// TIA Portal project "Tisch" (V17)

(* hardware
DEVICE "S7-1200-Station_2"  S7-1200 Station
   slot 0: "Baugruppenträger_0"  S7-1200 Rack  Rack  V1.0
   slot 1: "MTLab2-SPS-11"  CPU 1215C AC/DC/Rly  6ES7 215-1BG40-0XB0  V4.5
   slot 2: "DI 16/DQ 16x24VDC_1"  SM 1223 DI16/DQ16 x 24VDC  6ES7 223-1BL30-0XB0  V1.0
   slot 3: "DI 16/DQ 16x24VDC_2"  SM 1223 DI16/DQ16 x 24VDC  6ES7 223-1BL30-0XB0  V1.0
   slot 4: "AI 4x13BIT/AQ 2x14BIT_1"  SM 1234 AI4/AQ2  6ES7 234-4HE30-0XB0  V1.0
*)

// ===== PLC "MTLab2-SPS-11"  CPU 1215C AC/DC/Rly =====

VAR_GLOBAL   // PLC tag table "io_Tisch2_alt_Dreharm"
   "di_Encoder_ChA" AT %I0.0 : Bool;
   "di_Encoder_ChB" AT %I0.1 : Bool;
   "di_0Deg_Position" AT %I0.2 : Bool;
   "d_Z-Achse_ist_eingefahren" AT %I0.3 : Bool;
   "di_Z-Achse_ist_ausgefahren" AT %I0.4 : Bool;
   "di_Vertikalzylinder_ist_unten" AT %I0.5 : Bool;
   "di_Vertikalzylinder_ist_oben" AT %I0.6 : Bool;
   "do_Vertikalzylinder_nach_oben" AT %Q0.0 : Bool;
   "do_Sauger_ein" AT %Q0.1 : Bool;
   "do_Z-Achse_ausfahren" AT %Q0.2 : Bool;
   "do_drehen_links" AT %Q0.3 : Bool;
   "do_drehen_rechts" AT %Q0.4 : Bool;
   "di_Drehgeber_Wert" AT %ID1000 : DInt;
END_VAR

VAR_GLOBAL   // PLC tag table "io_Tisch2_alt_Förderband"
   "di_Lichtschranke" AT %E13.4 : Bool;
   "do_Rechtslauf" AT %A13.0 : Bool;
   "do_Linkslauf" AT %A13.1 : Bool;
END_VAR

VAR_GLOBAL   // PLC tag table "io_Tisch2_alt_Portal"
   "di_Zylinder_ist_oben" AT %E13.0 : Bool;
   "di_Zylinder_ist_unten" AT %E13.1 : Bool;
   "di_Shuttle_ist_rechts" AT %I13.2 : Bool;
   "di_Shuttle_ist_links" AT %I13.3 : Bool;
   "do_Zylinder_runter" AT %A8.4 : Bool;
   "do_Shuttle_links" AT %Q8.5 : Bool;
   "do_Saugen_ein" AT %Q8.6 : Bool;
END_VAR

VAR_GLOBAL   // PLC tag table "io_Tisch2_alt_Presse"
   "di_Sicherheitstür_ist_oben(1)" AT %E12.0 : Bool;
   "di_Sicherheitstür_ist_unten(1)" AT %E12.1 : Bool;
   "di_Ausschub_ist_ausgefahren(1)" AT %E12.2 : Bool;
   "di_Ausschub_ist_eingefahren(1)" AT %E12.3 : Bool;
   "di_Taster_rechts" AT %E12.4 : Bool;
   "di_Taster_links" AT %E12.5 : Bool;
   "do_Sicherheitstür_öffnen(1)" AT %A12.0 : Bool;
   "do_Sicherheitstür_schliessen(1)" AT %A12.1 : Bool;
   "do_Ausschub_ausfahren(1)" AT %A12.2 : Bool;
   "do_Ausschub_einfahren(1)" AT %A12.3 : Bool;
   "do_Lampe_rechts" AT %A12.4 : Bool;
   "do_Lampe_links" AT %A12.5 : Bool;
   "do_Stempel_senken(1)" AT %A12.6 : Bool;
   "do_Stempel_heben(1)" AT %A12.7 : Bool;
END_VAR

VAR_GLOBAL   // PLC tag table "io_Tisch2_alt_Stiftstation"
   "di_Klemmzylinder_ist_ausgefahren" AT %E1.1 : Bool;
   "di_Klemmzylinder_ist_eingefahren" AT %E1.2 : Bool;
   "di_Stiftzylinder_ist_ausgefahren" AT %E1.3 : Bool;
   "di_Stiftzylinder_ist_eingefahren" AT %E1.4 : Bool;
   "do_Klemmzylinder_ausfahren" AT %A0.7 : Bool;
   "do_Stiftzylinder_ausfahren" AT %A1.0 : Bool;
END_VAR

VAR_GLOBAL   // PLC tag table "io_Tisch2_alt_Bedienpult"
   "di_NotAus(NC)(1)" AT %E8.0 : Bool;
   "di_Hand(1)" AT %E8.1 : Bool;
   "di_Auto(1)" AT %E8.2 : Bool;
   "di_Start(1)" AT %E8.3 : Bool;
   "di_Stop(1)" AT %E8.4 : Bool;
   "di_Quit(1)" AT %E8.5 : Bool;
   "di_S6" AT %E8.6 : Bool;
   "di_NotAus(NO)" AT %E8.7 : Bool;
   "di_S1(1)" AT %E9.0 : Bool;
   "di_S2(1)" AT %E9.1 : Bool;
   "di_S3" AT %E9.2 : Bool;
   "di_S4" AT %E9.3 : Bool;
   "di_S5" AT %E9.4 : Bool;
   "do_Meldeleuchte_Bereit" AT %A8.0 : Bool;
   "do_Meldeleuchte_Läuft" AT %A8.1 : Bool;
   "do_Meldeleuchte_Fehler" AT %A8.2 : Bool;
   "do_Meldeleuchte_S6" AT %A8.3 : Bool;
END_VAR

TYPE "Type_Anlage"
   STRUCT
      Modus : Struct
         Grundstellung : Bool;
         Auto : Bool;
         Hand : Bool;
      END_STRUCT;
      NotHalt : Bool;
   END_STRUCT;
END_TYPE

TYPE "Type_Modul"
   STRUCT
      Kommando : Struct
         Start : Bool;
      END_STRUCT;
      Status : Struct
         Bereit : Bool;
         Fehler : Bool;
         LED : Bool;
      END_STRUCT;
      Parameter : Struct
         LongPressHomePosition : Time := T#2s;
      END_STRUCT;
   END_STRUCT;
END_TYPE

// folder: 1_DB

DATA_BLOCK "DB_Anlage"   // DB4
{ S7_Optimized_Access := 'TRUE' }
VERSION : 0.1
BEGIN
END_DATA_BLOCK

// folder: 8_Hardware/Aktoren

DATA_BLOCK "PortalLinks"   // DB25
{ S7_Optimized_Access := 'TRUE' }
VERSION : 0.1
// stored: InstanceOfName FB_SCL_Aktor
"FB_SCL_Aktor"
BEGIN
END_DATA_BLOCK

// folder: 8_Hardware/Sensoren

DATA_BLOCK "Starttaster"   // DB1
{ S7_Optimized_Access := 'TRUE' }
VERSION : 0.1
// stored: InstanceOfName FB_SCL_Sensor
"FB_SCL_Sensor"
BEGIN
END_DATA_BLOCK

DATA_BLOCK "Handmodus"   // DB2
{ S7_Optimized_Access := 'TRUE' }
VERSION : 0.1
// stored: InstanceOfName FB_SCL_Sensor
"FB_SCL_Sensor"
BEGIN
END_DATA_BLOCK

DATA_BLOCK "Automodus"   // DB3
{ S7_Optimized_Access := 'TRUE' }
VERSION : 0.1
// stored: InstanceOfName FB_SCL_Sensor
"FB_SCL_Sensor"
BEGIN
END_DATA_BLOCK

DATA_BLOCK "Grundstellung"   // DB5
{ S7_Optimized_Access := 'TRUE' }
VERSION : 0.1
// stored: InstanceOfName FB_SCL_Sensor
"FB_SCL_Sensor"
BEGIN
END_DATA_BLOCK

DATA_BLOCK "PortalBandseitig"   // DB21
{ S7_Optimized_Access := 'TRUE' }
VERSION : 0.1
// stored: InstanceOfName FB_SCL_Sensor
"FB_SCL_Sensor"
BEGIN
END_DATA_BLOCK

DATA_BLOCK "PortalPressenseitig"   // DB22
{ S7_Optimized_Access := 'TRUE' }
VERSION : 0.1
// stored: InstanceOfName FB_SCL_Sensor
"FB_SCL_Sensor"
BEGIN
END_DATA_BLOCK

DATA_BLOCK "PortalOben"   // DB23
{ S7_Optimized_Access := 'TRUE' }
VERSION : 0.1
// stored: InstanceOfName FB_SCL_Sensor
"FB_SCL_Sensor"
BEGIN
END_DATA_BLOCK

DATA_BLOCK "PortalUnten"   // DB24
{ S7_Optimized_Access := 'TRUE' }
VERSION : 0.1
// stored: InstanceOfName FB_SCL_Sensor
"FB_SCL_Sensor"
BEGIN
END_DATA_BLOCK

// folder: 8_Hardware/Zylinder

DATA_BLOCK "TestZylinder_1V2ES"   // DB20
{ S7_Optimized_Access := 'TRUE' }
VERSION : 0.1
// stored: InstanceOfName 1_FB_SCL_Zylinder_1V_2ES
"1_FB_SCL_Zylinder_1V_2ES"
BEGIN
END_DATA_BLOCK

// folder: 1_DB

FUNCTION "FC_Bedienpult" : Void   // FC4, FBD
{ S7_Optimized_Access := 'TRUE' }
VERSION : 0.1
BEGIN

REGION Network 1
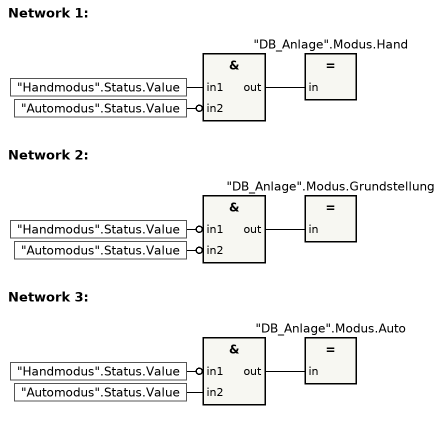
   "DB_Anlage".Modus.Hand := "Handmodus".Status.Value AND NOT "Automodus".Status.Value;
END_REGION

REGION Network 2
   "DB_Anlage".Modus.Grundstellung := NOT "Handmodus".Status.Value AND NOT "Automodus".Status.Value;
END_REGION

REGION Network 3
   "DB_Anlage".Modus.Auto := NOT "Handmodus".Status.Value AND "Automodus".Status.Value;
END_REGION
END_FUNCTION

ORGANIZATION_BLOCK "Main_DB"   // OB124, FBD, ProgramCycle
TITLE = "Main Program Sweep (Cycle)"
{ S7_Optimized_Access := 'TRUE' }
VERSION : 0.1
BEGIN

REGION Network 1: Variablen von/zum HMI aktualisieren
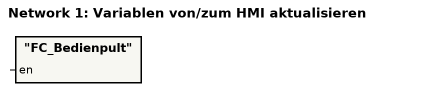
   "FC_Bedienpult"();
END_REGION
END_ORGANIZATION_BLOCK

// folder: 2_Ablauf/1_Module/4_Presse

FUNCTION_BLOCK "FB_SCL_Ablauf_Presse"   // FB8, SCL
{ S7_Optimized_Access := 'TRUE' }
VERSION : 0.1
   VAR_IN_OUT
      Zylinder_Ausschub : "0_FB_SCL_Zylinder_2V_2ES";
      Zylinder_Sicherheitstüre : "0_FB_SCL_Zylinder_2V_2ES";
      Zylinder_Presse : "0_FB_SCL_Zylinder_2V_2ES";
   END_VAR
   VAR
      homePosition : Bool;
      previousState : Int;
      currentState : Int;
      nextState : Int;
      stateStartTimeMs : UDInt;
      Kommando : Struct
         AutomatikStart : Bool;
         HomePositionStart : Bool;
         Retry : Bool;
      END_STRUCT;
      Status : Struct
         Ready : Bool;
         Error : Bool;
      END_STRUCT;
   END_VAR
   VAR_TEMP
      currentTimeMs : UDInt;
      stateActiveTimeS : UDInt;
      stateActiveTimeMs : UDInt;
   END_VAR
   VAR CONSTANT
      STATE_INIT : Int;
      STATE_READY : Int := 1;
      STATE_AUTO_FINISHED : Int := 2;
      STATE_AUTO_MOVE1 : Int := 3;
      STATE_HOMEPOSITION_FINISHED : Int := 4;
      STATE_HOMEPOSITION_MOVE1 : Int := 5;
      STATE_ERROR : Int := 6;
   END_VAR
BEGIN
   REGION State Machine Control
       // get current time
       "getTimestamp"(#currentTimeMs);

       REGION State Transition Check
           // check if a state transition is neccessary and store the time
           IF (#nextState <> #currentState) THEN
               // state transition occured!
               #previousState := #currentState;
               #currentState := #nextState;        // activate the new state
               #stateStartTimeMs := #currentTimeMs;  // store the time when the state was activated
           END_IF;
       END_REGION

       // calculate the time the state is already active
       #stateActiveTimeMs := #currentTimeMs - #stateStartTimeMs;
       #stateActiveTimeS := #stateActiveTimeMs / 1000;
   END_REGION


   // a move to startPosition request is executed regardless of the current state
   IF (#Kommando.HomePositionStart) THEN
       #nextState := #STATE_HOMEPOSITION_MOVE1;
   END_IF;

   REGION CASE Structure

       CASE #currentState OF


               // first state after machine startup
           #STATE_INIT:
               // set outputs to default values
               #Status.Ready := false;
               #Status.Error := false;

               // check if system is in "Grundstellung"
               IF (#homePosition) THEN
                   #nextState := #STATE_READY;
               END_IF;



           #STATE_READY:
               // system is ready to start
               #Status.Ready := true;

               // wait until rising edge of start signal occurs
               IF (#Kommando.AutomatikStart) THEN
                   #Status.Ready := false;
                   #nextState := #STATE_AUTO_MOVE1;
               END_IF;

           #STATE_AUTO_FINISHED:
               #nextState := #STATE_INIT;

           #STATE_HOMEPOSITION_FINISHED:
               #nextState := #STATE_INIT;




           #STATE_AUTO_MOVE1:
               // do something
               // 

               // if finished then goto finished
               #nextState := #STATE_AUTO_FINISHED;

               // transition to other states only if #DB_Anlage.Status.Auto_Aktiv is true!

           #STATE_HOMEPOSITION_MOVE1:
               // do something

               // if finished then goto finished
               #nextState := #STATE_HOMEPOSITION_FINISHED;

               // transition to other states only if #DB_Anlage.Status.Grundstellung_Aktiv is true!



           #STATE_ERROR:
               #Status.Ready := false;
               #Status.Error := true;

               // wait until the user has removed the error source
               IF (#Kommando.Retry) THEN
                   // go back to the last state and retry
                   #nextState := #previousState;
               END_IF;

       END_CASE;
   END_REGION

   // input signals are only true for one cycle
   #Kommando.AutomatikStart := false;
   #Kommando.HomePositionStart := false;
   #Kommando.Retry := false;
END_FUNCTION_BLOCK

// folder: 8_Hardware

FUNCTION "FC_Zylinder" : Void   // FC1, FBD
{ S7_Optimized_Access := 'TRUE' }
VERSION : 0.1
// hier werden den Zylindern die Ein- und Ausgänge zugewiesen
BEGIN

REGION Network 1
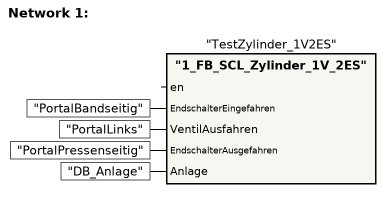
   "TestZylinder_1V2ES"(EndschalterEingefahren := "PortalBandseitig",   // "1_FB_SCL_Zylinder_1V_2ES"
                        VentilAusfahren := "PortalLinks",
                        EndschalterAusgefahren := "PortalPressenseitig",
                        Anlage := "DB_Anlage");
END_REGION
END_FUNCTION

FUNCTION "FC_Aktoren" : Void   // FC2, FBD
{ S7_Optimized_Access := 'TRUE' }
VERSION : 0.1
BEGIN

REGION Network 1
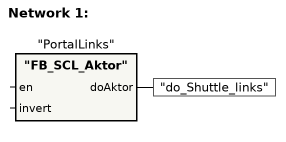
   "PortalLinks"(doAktor => "do_Shuttle_links");   // "FB_SCL_Aktor"
END_REGION
END_FUNCTION

FUNCTION "FC_Sensor" : Void   // FC3, FBD
{ S7_Optimized_Access := 'TRUE' }
VERSION : 0.1
BEGIN

REGION Network 1
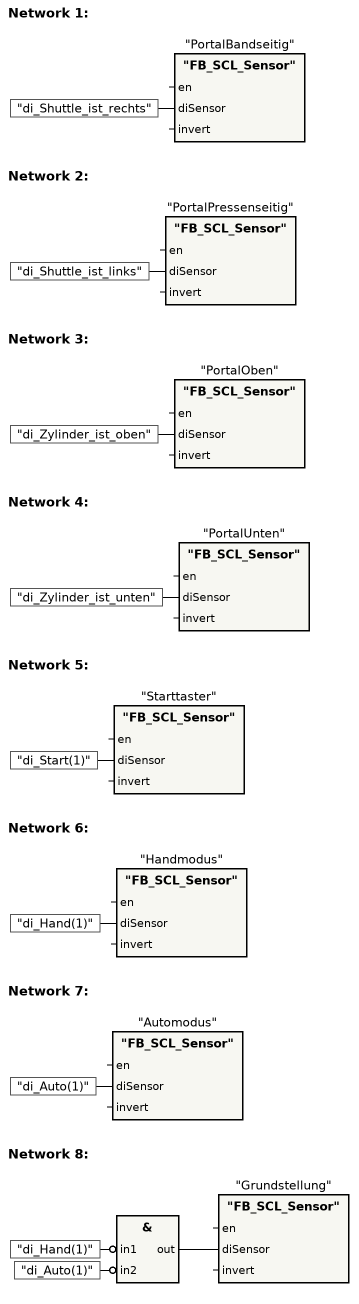
   "PortalBandseitig"(diSensor := "di_Shuttle_ist_rechts");   // "FB_SCL_Sensor"
END_REGION

REGION Network 2
   "PortalPressenseitig"(diSensor := "di_Shuttle_ist_links");   // "FB_SCL_Sensor"
END_REGION

REGION Network 3
   "PortalOben"(diSensor := "di_Zylinder_ist_oben");   // "FB_SCL_Sensor"
END_REGION

REGION Network 4
   "PortalUnten"(diSensor := "di_Zylinder_ist_unten");   // "FB_SCL_Sensor"
END_REGION

REGION Network 5
   "Starttaster"(diSensor := "di_Start(1)");   // "FB_SCL_Sensor"
END_REGION

REGION Network 6
   "Handmodus"(diSensor := "di_Hand(1)");   // "FB_SCL_Sensor"
END_REGION

REGION Network 7
   "Automodus"(diSensor := "di_Auto(1)");   // "FB_SCL_Sensor"
END_REGION

REGION Network 8
   "Grundstellung"(diSensor := NOT "di_Hand(1)" AND NOT "di_Auto(1)");   // "FB_SCL_Sensor"
END_REGION
END_FUNCTION

ORGANIZATION_BLOCK "Main_Hardware"   // OB123, FBD, ProgramCycle
TITLE = "Main Program Sweep (Cycle)"
{ S7_Optimized_Access := 'TRUE' }
VERSION : 0.1
BEGIN

REGION Network 1: Motoren ansteuern
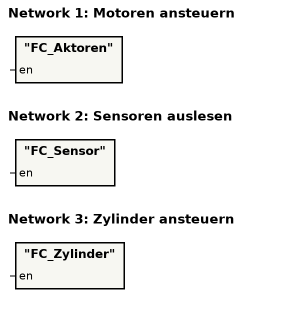
   "FC_Aktoren"();
END_REGION

REGION Network 2: Sensoren auslesen
   "FC_Sensor"();
END_REGION

REGION Network 3: Zylinder ansteuern
   "FC_Zylinder"();
END_REGION
END_ORGANIZATION_BLOCK

// folder: 9_Lib/0_Hardware/Sensor

FUNCTION_BLOCK "FB_SCL_Sensor"   // FB3, SCL
{ S7_Optimized_Access := 'TRUE' }
VERSION : 0.1
   VAR_INPUT
      diSensor : Bool;
      invert : Bool;
   END_VAR
   VAR
      Status : Struct
         Value : Bool;
      END_STRUCT;
   END_VAR
BEGIN
   IF #invert = TRUE THEN          //If Value is inverted, then return the inverted value
       #Status.Value := NOT #diSensor;
   ELSE                            //If Value is not inverted, then return the value itself
       #Status.Value := #diSensor;
   END_IF;
END_FUNCTION_BLOCK

FUNCTION_BLOCK "FB_SCL_Aktor"   // FB5, SCL
{ S7_Optimized_Access := 'TRUE' }
VERSION : 0.1
   VAR_INPUT
      invert : Bool;
   END_VAR
   VAR_OUTPUT
      doAktor : Bool;
   END_VAR
   VAR
      Kommando : Struct
         Value : Bool;
      END_STRUCT;
   END_VAR
BEGIN
   IF #invert THEN
       #doAktor := NOT #Kommando.Value;
   ELSE
       #doAktor := #Kommando.Value;
   END_IF;
END_FUNCTION_BLOCK

// folder: 9_Lib/0_Hardware/Zylinder/Varianten

FUNCTION_BLOCK "0_FB_SCL_Zylinder_2V_2ES"   // FB1, SCL
{ S7_Optimized_Access := 'TRUE' }
VERSION : 0.1
   VAR_IN_OUT
      EndschalterEingefahren : "FB_SCL_Sensor";
      VentilAusfahren : "FB_SCL_Aktor";
      VentilEinfahren : "FB_SCL_Aktor";
      EndschalterAusgefahren : "FB_SCL_Sensor";
      Anlage : "Type_Anlage";
   END_VAR
   VAR
      Status : Struct
         istAusgefahren : Bool;
         istEingefahren : Bool;
         Fehler : Bool;
         Bereit : Bool;
      END_STRUCT;
      Parameter : Struct
         timeoutEinfahrenMS : Int := 1000;
         timeoutAusfahrenMS : Int := 1000;
         ZeitDruckaufbauMS : Int := 250;
         WartezeitInitMS : Int := 250;
      END_STRUCT;
      Kommando : Struct
         einfahren : Bool;
         ausfahren : Bool;
         einzelschrittStart : Bool;
      END_STRUCT;
      StateMachine : Struct
         CurrentState : Int := 999;
         NextState : Int;
         StateStartTimeMS : UDInt;
      END_STRUCT;
   END_VAR
   VAR_TEMP
      CurrentTimeMS : UDInt;
      stateActiveTimeMS : UDInt;
   END_VAR
   VAR CONSTANT
      STATE_INIT : Int := 0;
      STATE_BUILDPRESSURE : Int := 1;
      STATE_READY : Int := 2;
      STATE_SINGLEEXTEND : Int := 3;
      STATE_EXTEND : Int := 4;
      STATE_ENDPOS : Int := 5;
      STATE_ERROR : Int := 6;
      STATE_SINGLERETRACT : Int := 7;
      STATE_RETRACT : Int := 8;
   END_VAR
BEGIN
   REGION NotHalt

       IF #Anlage.NotHalt THEN
           #VentilAusfahren.Kommando.Value := FALSE;
           #VentilEinfahren.Kommando.Value := FALSE;
           RETURN;
       END_IF;

   END_REGION

   REGION Timing
       // get current time
       "getTimestamp"(#CurrentTimeMS);


       // check if a state transition is neccessary and store the time
       IF (#StateMachine.NextState <> #StateMachine.CurrentState) THEN
           // state transition occured!
           #StateMachine.CurrentState := #StateMachine.NextState;        // activate the new state
           #StateMachine.StateStartTimeMS := #CurrentTimeMS;  // store the time when the state was activated
       END_IF;

       // calculate the time the state is already active
       #stateActiveTimeMS := #CurrentTimeMS - #StateMachine.StateStartTimeMS;
   END_REGION

   REGION Logik

       CASE #StateMachine.CurrentState OF

           #STATE_INIT:  //INIT
               REGION INIT

               IF #stateActiveTimeMS > #Parameter.WartezeitInitMS THEN
                   #StateMachine.NextState := #STATE_BUILDPRESSURE;
               END_IF;
           END_REGION

           #STATE_BUILDPRESSURE:
               REGION BUILD PRESSURE
               #Status.Fehler := FALSE;

               IF (#EndschalterAusgefahren.Status.Value AND #EndschalterEingefahren.Status.Value) OR (NOT #EndschalterAusgefahren.Status.Value AND NOT #EndschalterEingefahren.Status.Value) THEN
                   #Status.Fehler := TRUE;
                   #VentilEinfahren.Kommando.Value := false;
                   #VentilAusfahren.Kommando.Value := false;
                   #StateMachine.NextState := #STATE_READY;
               END_IF;

               IF #EndschalterAusgefahren.Status.Value AND NOT #EndschalterEingefahren.Status.Value THEN
                   #VentilAusfahren.Kommando.Value := true;
                   #VentilEinfahren.Kommando.Value := false;
               ELSIF #EndschalterEingefahren.Status.Value AND NOT #EndschalterAusgefahren.Status.Value THEN
                   #VentilAusfahren.Kommando.Value := FALSE;
                   #VentilEinfahren.Kommando.Value := TRUE;
               END_IF;

               IF #stateActiveTimeMS > #Parameter.ZeitDruckaufbauMS THEN
                   #VentilEinfahren.Kommando.Value := false;
                   #VentilAusfahren.Kommando.Value := false;
                   #StateMachine.NextState := #STATE_READY;
               END_IF;

           END_REGION

           #STATE_READY:
               REGION Ready
                   #Status.Bereit := true;
                   IF #Kommando.ausfahren AND NOT #VentilAusfahren.Kommando.Value THEN
                       #StateMachine.NextState := #STATE_SINGLEEXTEND;
                   END_IF;

                   IF #Kommando.einfahren AND NOT #EndschalterEingefahren.Status.Value THEN
                       #StateMachine.NextState := #STATE_SINGLERETRACT;
                   END_IF;

               END_REGION

           #STATE_SINGLEEXTEND:
               REGION Single Step Extension

                   #Status.Bereit := false;

                   IF NOT #Anlage.Modus.Hand THEN
                       #StateMachine.NextState := #STATE_READY;
                   END_IF;

                   IF #Anlage.Modus.Hand AND #Kommando.einzelschrittStart THEN
                       #StateMachine.NextState := #STATE_EXTEND;
                   END_IF;

                   IF #Anlage.Modus.Auto OR #Anlage.Modus.Grundstellung THEN
                       #StateMachine.NextState := #STATE_EXTEND;
                   END_IF;

               END_REGION

           #STATE_EXTEND:
               REGION Extension
                   #VentilAusfahren.Kommando.Value := true;
                   IF #EndschalterAusgefahren.Status.Value THEN
                       #StateMachine.NextState := #STATE_ENDPOS;
                   END_IF;

                   IF #stateActiveTimeMS > #Parameter.timeoutAusfahrenMS THEN
                       #StateMachine.NextState := #STATE_ERROR;
                   END_IF;
               END_REGION;

           #STATE_SINGLERETRACT:
               REGION Single Step Retract

                   #Status.Bereit := false;

                   IF NOT #Anlage.Modus.Hand THEN
                       #StateMachine.NextState := #STATE_READY;
                   END_IF;

                   IF #Anlage.Modus.Hand AND #Kommando.einzelschrittStart THEN
                       #StateMachine.NextState := #STATE_RETRACT;
                   END_IF;

                   IF #Anlage.Modus.Auto OR #Anlage.Modus.Grundstellung THEN
                       #StateMachine.NextState := #STATE_RETRACT;
                   END_IF;

               END_REGION

           #STATE_RETRACT:
               REGION Extension
                   #VentilEinfahren.Kommando.Value := true;
                   IF #EndschalterEingefahren.Status.Value THEN
                       #StateMachine.NextState := #STATE_ENDPOS;
                   END_IF;

                   IF #stateActiveTimeMS > #Parameter.timeoutEinfahrenMS THEN
                       #StateMachine.NextState := #STATE_ERROR;
                   END_IF;
               END_REGION

           #STATE_ENDPOS:
               REGION End Position
                   #VentilAusfahren.Kommando.Value := false;
                   #VentilEinfahren.Kommando.Value := false;
                   #Status.Fehler := false;
                   #StateMachine.NextState := #STATE_READY;
               END_REGION;

           #STATE_ERROR:
               REGION End Position
                   #VentilAusfahren.Kommando.Value := false;
                   #VentilEinfahren.Kommando.Value := false;
                   #Status.Fehler := true;
                   #StateMachine.NextState := #STATE_READY;
               END_REGION ;


       END_CASE;


   END_REGION

   REGION KommandoReset

       #Kommando.ausfahren := FALSE;
       #Kommando.einfahren := FALSE;
       #Kommando.einzelschrittStart := FALSE;

   END_REGION
END_FUNCTION_BLOCK

FUNCTION_BLOCK "1_FB_SCL_Zylinder_1V_2ES"   // FB2, SCL
{ S7_Optimized_Access := 'TRUE' }
VERSION : 0.1
   VAR_IN_OUT
      EndschalterEingefahren : "FB_SCL_Sensor";
      VentilAusfahren : "FB_SCL_Aktor";
      EndschalterAusgefahren : "FB_SCL_Sensor";
      Anlage : "Type_Anlage";
   END_VAR
   VAR
      Status : Struct
         istAusgefahren : Bool;
         istEingefahren : Bool;
         Fehler : Bool;
         Bereit : Bool;
      END_STRUCT;
      Parameter : Struct
         timeoutEinfahrenMS : Int := 1000;
         timeoutAusfahrenMS : Int := 1000;
         ZeitDruckaufbauMS : Int := 250;
         WartezeitInitMS : Int := 250;
      END_STRUCT;
      Kommando : Struct
         einfahren : Bool;
         ausfahren : Bool;
         einzelschrittStart : Bool;
      END_STRUCT;
      StaticOutput : Bool;   // Static Variable to set for output
      StateMachine : Struct
         CurrentState : Int := 999;
         NextState : Int;
         StateStartTimeMS : UDInt;
      END_STRUCT;
   END_VAR
   VAR_TEMP
      CurrentTimeMS : UDInt;
      stateActiveTimeMS : UDInt;
   END_VAR
   VAR CONSTANT
      STATE_INIT : Int := 0;
      STATE_BUILDPRESSURE : Int := 1;
      STATE_READY : Int := 2;
      STATE_SINGLEEXTEND : Int := 3;
      STATE_EXTEND : Int := 4;
      STATE_ENDPOS : Int := 5;
      STATE_ERROR : Int := 6;
      STATE_SINGLERETRACT : Int := 7;
      STATE_RETRACT : Int := 8;
   END_VAR
BEGIN
   //Copied code from 0_FB_SCL_Zylinder_2V_2ES,
   //Output is now a static variable ("StaticOutput"), which is written to the output at the end
   //There is no Valve for Contraction

   REGION NotHalt

       IF #Anlage.NotHalt THEN
           #VentilAusfahren.Kommando.Value := FALSE;
           RETURN;
       END_IF;

   END_REGION

   REGION Timing
       // get current time
       "getTimestamp"(#CurrentTimeMS);


       // check if a state transition is neccessary and store the time
       IF (#StateMachine.NextState <> #StateMachine.CurrentState) THEN
           // state transition occured!
           #StateMachine.CurrentState := #StateMachine.NextState;        // activate the new state
           #StateMachine.StateStartTimeMS := #CurrentTimeMS;  // store the time when the state was activated
       END_IF;

       // calculate the time the state is already active
       #stateActiveTimeMS := #CurrentTimeMS - #StateMachine.StateStartTimeMS;
   END_REGION

   REGION Logik

       CASE #StateMachine.CurrentState OF

           #STATE_INIT:  //INIT
               REGION INIT

               IF #stateActiveTimeMS > #Parameter.WartezeitInitMS THEN
                   #StateMachine.NextState := #STATE_BUILDPRESSURE;
               END_IF;
           END_REGION

           #STATE_BUILDPRESSURE:
               REGION BUILD PRESSURE
               #Status.Fehler := FALSE;

               IF (#EndschalterAusgefahren.Status.Value AND #EndschalterEingefahren.Status.Value) OR (NOT #EndschalterAusgefahren.Status.Value AND NOT #EndschalterEingefahren.Status.Value) THEN
                   #Status.Fehler := TRUE;
                   #StaticOutput := FALSE;
                   #StateMachine.NextState := #STATE_READY;
               END_IF;

               IF #EndschalterAusgefahren.Status.Value AND NOT #EndschalterEingefahren.Status.Value THEN
                   #StaticOutput := TRUE;
               ELSIF #EndschalterEingefahren.Status.Value AND NOT #EndschalterAusgefahren.Status.Value THEN
                   #StaticOutput := FALSE;
               END_IF;

               IF #stateActiveTimeMS > #Parameter.ZeitDruckaufbauMS THEN
                   #StaticOutput := FALSE;
                   #StateMachine.NextState := #STATE_READY;
               END_IF;

           END_REGION

           #STATE_READY:
               REGION Ready
                   #Status.Bereit := true;
                   IF #Kommando.ausfahren AND NOT #VentilAusfahren.Kommando.Value THEN
                       #StateMachine.NextState := #STATE_SINGLEEXTEND;
                   END_IF;

                   IF #Kommando.einfahren AND NOT #EndschalterEingefahren.Status.Value THEN
                       #StateMachine.NextState := #STATE_SINGLERETRACT;
                   END_IF;

               END_REGION

           #STATE_SINGLEEXTEND:
               REGION Single Step Extension

                   #Status.Bereit := false;

                   IF NOT #Anlage.Modus.Hand THEN
                       #StateMachine.NextState := #STATE_READY;
                   END_IF;

                   IF #Anlage.Modus.Hand AND #Kommando.einzelschrittStart THEN
                       #StateMachine.NextState := #STATE_EXTEND;
                   END_IF;

                   IF #Anlage.Modus.Auto OR #Anlage.Modus.Grundstellung THEN
                       #StateMachine.NextState := #STATE_EXTEND;
                   END_IF;

               END_REGION

           #STATE_EXTEND:
               REGION Extension
                   //Extend
                   #StaticOutput := TRUE;
                   IF #EndschalterAusgefahren.Status.Value THEN
                       #StateMachine.NextState := #STATE_ENDPOS;
                   END_IF;

                   IF #stateActiveTimeMS > #Parameter.timeoutAusfahrenMS THEN
                       #StateMachine.NextState := #STATE_ERROR;
                   END_IF;
               END_REGION;

           #STATE_SINGLERETRACT:
               REGION Single Step Retract

                   #Status.Bereit := false;

                   IF NOT #Anlage.Modus.Hand THEN
                       #StateMachine.NextState := #STATE_READY;
                   END_IF;

                   IF #Anlage.Modus.Hand AND #Kommando.einzelschrittStart THEN
                       #StateMachine.NextState := #STATE_RETRACT;
                   END_IF;

                   IF #Anlage.Modus.Auto OR #Anlage.Modus.Grundstellung THEN
                       #StateMachine.NextState := #STATE_RETRACT;
                   END_IF;

               END_REGION

           #STATE_RETRACT:
               REGION Retraction
                   //Retract
                   #StaticOutput := FALSE;
                   IF #EndschalterEingefahren.Status.Value THEN
                       #StateMachine.NextState := #STATE_ENDPOS;
                   END_IF;

                   IF #stateActiveTimeMS > #Parameter.timeoutEinfahrenMS THEN
                       #StateMachine.NextState := #STATE_ERROR;
                   END_IF;
               END_REGION

           #STATE_ENDPOS:
               REGION End Position
                   #Status.Fehler := false;
                   #StateMachine.NextState := #STATE_READY;
               END_REGION;

           #STATE_ERROR:
               REGION End Position
                   //Do not change output, as a change would generate movement
                   #Status.Fehler := true;
                   #StateMachine.NextState := #STATE_READY;
               END_REGION ;


       END_CASE;


   END_REGION

   REGION KommandoReset

       #Kommando.ausfahren := FALSE;
       #Kommando.einfahren := FALSE;
       #Kommando.einzelschrittStart := FALSE;

   END_REGION

   REGION Output
       #VentilAusfahren.Kommando.Value := #StaticOutput;
       #Status.istAusgefahren := #EndschalterAusgefahren.Status.Value;
       #Status.istEingefahren := #EndschalterEingefahren.Status.Value;
   END_REGION
END_FUNCTION_BLOCK

FUNCTION_BLOCK "FB_Zylinder"   // FB7, FBD
{ S7_Optimized_Access := 'TRUE' }
VERSION : 0.1
   VAR_INPUT
      AnzahlEndschalter : Int := 2;
      AnzahlVentile : Int := 2;
   END_VAR
   VAR_IN_OUT
      VentilAusfahren : "FB_SCL_Aktor";
      EndschalterEingefahren : "FB_SCL_Sensor";
      VentilEinfahren : "FB_SCL_Aktor";
      EndschalterAusgefahren : "FB_SCL_Sensor";
      Anlage : "Type_Anlage";
   END_VAR
   VAR
      "2V2ES" : "0_FB_SCL_Zylinder_2V_2ES";
      "1V2ES" : "1_FB_SCL_Zylinder_1V_2ES";
   END_VAR
BEGIN

REGION Network 1
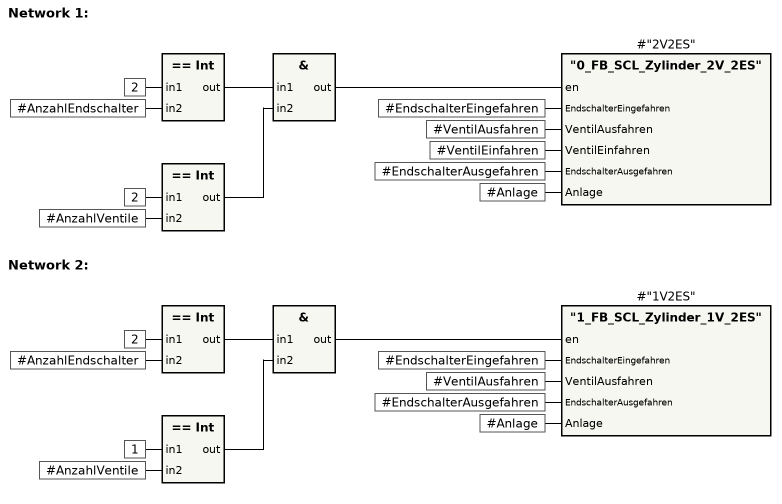
   IF (2 = #AnzahlEndschalter) AND (2 = #AnzahlVentile) THEN
       #"2V2ES"(EndschalterEingefahren := #EndschalterEingefahren,   // "0_FB_SCL_Zylinder_2V_2ES"
                VentilAusfahren := #VentilAusfahren,
                VentilEinfahren := #VentilEinfahren,
                EndschalterAusgefahren := #EndschalterAusgefahren,
                Anlage := #Anlage);
   END_IF;
END_REGION

REGION Network 2
   IF (2 = #AnzahlEndschalter) AND (1 = #AnzahlVentile) THEN
       #"1V2ES"(EndschalterEingefahren := #EndschalterEingefahren,   // "1_FB_SCL_Zylinder_1V_2ES"
                VentilAusfahren := #VentilAusfahren,
                EndschalterAusgefahren := #EndschalterAusgefahren,
                Anlage := #Anlage);
   END_IF;
END_REGION
END_FUNCTION_BLOCK

// folder: 9_Lib/1_Funktionen

FUNCTION "getTimestamp" : Void   // FC5, SCL
{ S7_Optimized_Access := 'TRUE' }
VERSION : 0.1
   VAR_OUTPUT
      TS_OUT : UDInt;
   END_VAR
   VAR_TEMP
      actDT : DTL;
      tmp : Int;
   END_VAR
BEGIN
   // Uhrzeit lesen
   #tmp := RD_SYS_T(OUT => #actDT);

   // in Timestamp konvertieren (Quelle: https://support.industry.siemens.com/forum/at/en/posts/s7-1200-unix-timestamp/108455)
   #TS_OUT := (DATE_TO_UDINT(DTL_TO_DATE(#actDT)) * 86400000) + (TOD_TO_UDINT(DTL_TO_TOD(#actDT))) + 631152000; //TS as UDINT
END_FUNCTION

// folder: 9_Lib/9_Vorlagen

FUNCTION_BLOCK "FB_SCL_Vorlage_ModulLogik"   // FB4, SCL
{ S7_Optimized_Access := 'TRUE' }
VERSION : 0.1
   VAR_IN_OUT
      DB_Modul : "Type_Modul";
      DB_Anlage : "Type_Anlage";
   END_VAR
   VAR
      TON_HomePosition : TON_TIME;
   END_VAR
   VAR_TEMP
      HomePositionStart : Bool;
      AutoStart : Bool;
   END_VAR
BEGIN
   REGION Init
       #HomePositionStart := false;
   END_REGION


   REGION Signal Processing

       REGION Home Position Request

           #TON_HomePosition(IN := #DB_Modul.Kommando.Start,
                             PT := #DB_Modul.Parameter.LongPressHomePosition);
           IF #DB_Anlage.Modus.Grundstellung AND #TON_HomePosition.Q THEN
               #HomePositionStart := true;
           END_IF;


       END_REGION



   END_REGION
END_FUNCTION_BLOCK

FUNCTION_BLOCK "FB_SCL_Vorlage_ModulAblauf"   // FB6, SCL
{ S7_Optimized_Access := 'TRUE' }
VERSION : 0.1
   VAR
      homePosition : Bool;
      previousState : Int;
      currentState : Int;
      nextState : Int;
      stateStartTimeMs : UDInt;
      Kommando : Struct
         AutomatikStart : Bool;
         HomePositionStart : Bool;
         Retry : Bool;
      END_STRUCT;
      Status : Struct
         Ready : Bool;
         Error : Bool;
      END_STRUCT;
   END_VAR
   VAR_TEMP
      currentTimeMs : UDInt;
      stateActiveTimeS : UDInt;
      stateActiveTimeMs : UDInt;
   END_VAR
   VAR CONSTANT
      STATE_INIT : Int;
      STATE_READY : Int := 1;
      STATE_AUTO_FINISHED : Int := 2;
      STATE_AUTO_MOVE1 : Int := 3;
      STATE_HOMEPOSITION_FINISHED : Int := 4;
      STATE_HOMEPOSITION_MOVE1 : Int := 5;
      STATE_ERROR : Int := 6;
   END_VAR
BEGIN
   REGION State Machine Control
       // get current time
       "getTimestamp"(#currentTimeMs);

       REGION State Transition Check
           // check if a state transition is neccessary and store the time
           IF (#nextState <> #currentState) THEN
               // state transition occured!
               #previousState := #currentState;
               #currentState := #nextState;        // activate the new state
               #stateStartTimeMs := #currentTimeMs;  // store the time when the state was activated
           END_IF;
       END_REGION

       // calculate the time the state is already active
       #stateActiveTimeMs := #currentTimeMs - #stateStartTimeMs;
       #stateActiveTimeS := #stateActiveTimeMs / 1000;
   END_REGION


   // a move to startPosition request is executed regardless of the current state
   IF (#Kommando.HomePositionStart) THEN
       #nextState := #STATE_HOMEPOSITION_MOVE1;
   END_IF;

   REGION CASE Structure

       CASE #currentState OF


               // first state after machine startup
           #STATE_INIT:
               // set outputs to default values
               #Status.Ready := false;
               #Status.Error := false;

               // check if system is in "Grundstellung"
               IF (#homePosition) THEN
                   #nextState := #STATE_READY;
               END_IF;



           #STATE_READY:
               // system is ready to start
               #Status.Ready := true;

               // wait until rising edge of start signal occurs
               IF (#Kommando.AutomatikStart) THEN
                   #Status.Ready := false;
                   #nextState := #STATE_AUTO_MOVE1;
               END_IF;

           #STATE_AUTO_FINISHED:
               #nextState := #STATE_INIT;

           #STATE_HOMEPOSITION_FINISHED:
               #nextState := #STATE_INIT;




           #STATE_AUTO_MOVE1:
               // do something
               // 

               // if finished then goto finished
               #nextState := #STATE_AUTO_FINISHED;

               // transition to other states only if #DB_Anlage.Status.Auto_Aktiv is true!

           #STATE_HOMEPOSITION_MOVE1:
               // do something

               // if finished then goto finished
               #nextState := #STATE_HOMEPOSITION_FINISHED;

               // transition to other states only if #DB_Anlage.Status.Grundstellung_Aktiv is true!



           #STATE_ERROR:
               #Status.Ready := false;
               #Status.Error := true;

               // wait until the user has removed the error source
               IF (#Kommando.Retry) THEN
                   // go back to the last state and retry
                   #nextState := #previousState;
               END_IF;

       END_CASE;
   END_REGION

   // input signals are only true for one cycle
   #Kommando.AutomatikStart := false;
   #Kommando.HomePositionStart := false;
   #Kommando.Retry := false;
END_FUNCTION_BLOCK